FUNCTION_BLOCK ELLIP_ENVELOPE
  {SET_ATTRIBUTE(OpcUa, SERVICE)}
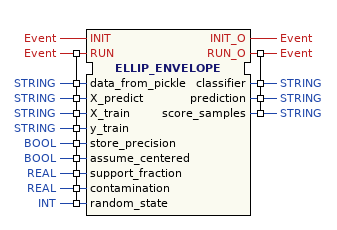
  EVENT_INPUT
    INIT;
    RUN WITH data_from_pickle, X_predict, X_train, y_train, store_precision, assume_centered, support_fraction, contamination, random_state; {SET_ATTRIBUTE(OpcUa, Method)}
  END_EVENT
  EVENT_OUTPUT
    INIT_O;
    RUN_O WITH classifier, prediction, score_samples;
  END_EVENT
  VAR_INPUT
    data_from_pickle : STRING; {SET_ATTRIBUTE(OpcUa, Variable.RUN)}
    X_predict : STRING; {SET_ATTRIBUTE(OpcUa, Variable.RUN)}
    X_train : STRING; {SET_ATTRIBUTE(OpcUa, Variable.RUN)}
    y_train : STRING; {SET_ATTRIBUTE(OpcUa, Variable.RUN)}
    store_precision : BOOL; {SET_ATTRIBUTE(OpcUa, Variable.RUN)}
    assume_centered : BOOL; {SET_ATTRIBUTE(OpcUa, Variable.RUN)}
    support_fraction : REAL; {SET_ATTRIBUTE(OpcUa, Variable.RUN)}
    contamination : REAL; {SET_ATTRIBUTE(OpcUa, Variable.RUN)}
    random_state : INT; {SET_ATTRIBUTE(OpcUa, Variable.RUN)}
  END_VAR
  VAR_OUTPUT
    classifier : STRING; {SET_ATTRIBUTE(OpcUa, Variable.RUN)}
    prediction : STRING; {SET_ATTRIBUTE(OpcUa, Variable.RUN)}
    score_samples : STRING; {SET_ATTRIBUTE(OpcUa, Variable.RUN)}
  END_VAR
END_FUNCTION_BLOCK
